FUNCTION_BLOCK BYPASS_AX_BOOL (* Bypass FB *)
  (* Standard: 61499-2 *)
  (* Version 1.0, 2026-05-07, franz *)
  PACKAGE logiBUS::signalprocessing::bypass;
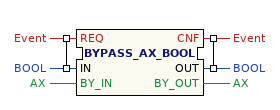
  EVENT_INPUT
    REQ WITH IN; (* Normal Execution Request *)
  END_EVENT
  EVENT_OUTPUT
    CNF WITH OUT; (* Execution Confirmation *)
  END_EVENT
  VAR_INPUT
    IN : BOOL; (* Input *)
  END_VAR
  VAR_OUTPUT
    OUT : BOOL; (* Output *)
  END_VAR
  SOCKETS
    BY_IN : adapter::types::unidirectional::AX; (* Bypass in *)
  END_SOCKETS
  PLUGS
    BY_OUT : adapter::types::unidirectional::AX; (* Bypass out *)
  END_PLUGS
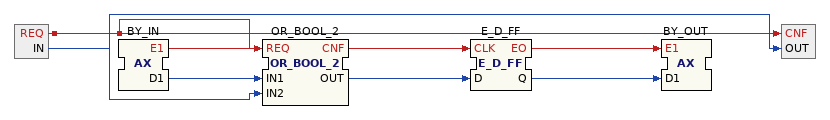
  FBS
    OR_BOOL_2 : iec61131::booleanOperators::OR_BOOL_2;
    E_D_FF : iec61499::events::E_D_FF;
  END_FBS
  EVENT_CONNECTIONS
    OR_BOOL_2.CNF TO E_D_FF.CLK;
    BY_IN.E1 TO OR_BOOL_2.REQ;
    E_D_FF.EO TO BY_OUT.E1;
    REQ TO CNF;
    REQ TO OR_BOOL_2.REQ;
  END_CONNECTIONS
  DATA_CONNECTIONS
    OR_BOOL_2.OUT TO E_D_FF.D;
    BY_IN.D1 TO OR_BOOL_2.IN1;
    E_D_FF.Q TO BY_OUT.D1;
    IN TO OUT;
    IN TO OR_BOOL_2.IN2;
  END_CONNECTIONS
END_FUNCTION_BLOCK
